FUNCTION_BLOCK setTimers (* Composite Function Block Type *)
  (* Standard: 61499-2 *)
  (* Version 0.2, 2003-12-05, JHC, Rockwell Automation, Renamed from NEWCOMPFB. *)
  (* Version 0.1, 2002-01-08, JHC, Rockwell Automation, Added DLY FB as example. *)
  (* Version 0.0, 2000-05-27, JHC, Rockwell Automation *)
  (* Compiler header: package fb.rt.template; *)
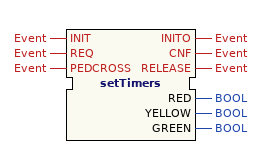
  EVENT_INPUT
    INIT; (* Initialization Request *)
    REQ; (* Normal Execution Request *)
    PEDCROSS;
  END_EVENT
  EVENT_OUTPUT
    INITO; (* Initialization Confirm *)
    CNF; (* Execution Confirmation *)
    RELEASE;
  END_EVENT
  VAR_OUTPUT
    RED : BOOL;
    YELLOW : BOOL;
    GREEN : BOOL;
  END_VAR
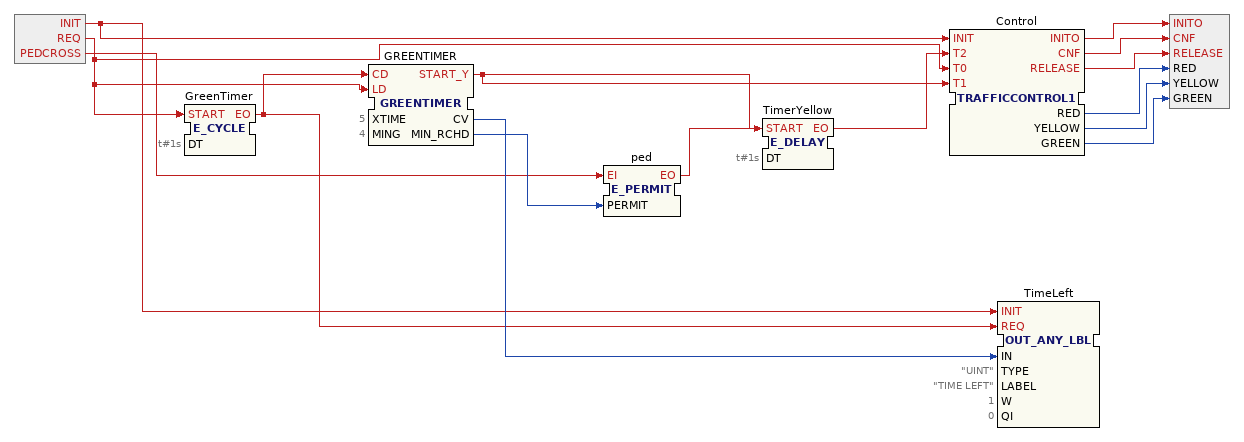
  FBS
    Control : TRAFFICCONTROL1;
    TimerYellow : E_DELAY(DT := t#1s);
    TimeLeft : OUT_ANY_LBL(TYPE := "UINT", LABEL := "TIME LEFT", W := 1, QI := 0);
    GreenTimer : E_CYCLE(DT := t#1s);
    ped : E_PERMIT;
    GREENTIMER : GREENTIMER(XTIME := 5, MING := 4);
  END_FBS
  EVENT_CONNECTIONS
    INIT TO Control.INIT;
    TimerYellow.EO TO Control.T2;
    Control.INITO TO INITO;
    Control.CNF TO CNF;
    REQ TO Control.T0;
    Control.RELEASE TO RELEASE;
    INIT TO TimeLeft.INIT;
    REQ TO GreenTimer.START;
    PEDCROSS TO ped.EI;
    ped.EO TO TimerYellow.START;
    GreenTimer.EO TO GREENTIMER.CD;
    GREENTIMER.START_Y TO Control.T1;
    GREENTIMER.START_Y TO TimerYellow.START;
    GreenTimer.EO TO TimeLeft.REQ;
    REQ TO GREENTIMER.LD;
  END_CONNECTIONS
  DATA_CONNECTIONS
    Control.RED TO RED;
    Control.YELLOW TO YELLOW;
    Control.GREEN TO GREEN;
    GREENTIMER.CV TO TimeLeft.IN;
    GREENTIMER.MIN_RCHD TO ped.PERMIT;
  END_CONNECTIONS
END_FUNCTION_BLOCK
